{attribute 'qualified_only'}
VAR_GLOBAL CONSTANT
	CNUM_AXIS : INT := 3;
END_VAR

(* stored: Version 1.1.0.1, ProductVersion 3.1.4024.16
   GVL GVL_MotorControl: Id {6d3ad16d-b7c0-47e1-82ea-bcdc2426d51a} *)
